FUNCTION_BLOCK BasicAdapter2 (* Basic FB with empty ECC *)
  (* Standard: 61499-2 *)
  (* Version 1.0, 2023-03-07, AK115394 *)
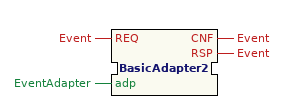
  EVENT_INPUT
    REQ;
  END_EVENT
  EVENT_OUTPUT
    CNF;
    RSP;
  END_EVENT
  SOCKETS
    adp : EventAdapter;
  END_SOCKETS
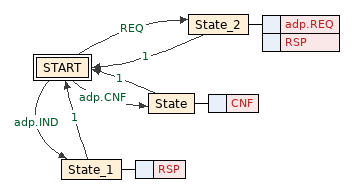
  EC_STATES
    START; (* Initial State *)
    State_2 : -> adp.REQ, -> RSP;
    State : -> CNF;
    State_1 : -> RSP;
  END_STATES
  EC_TRANSITIONS
    START TO State_2 := REQ;
    State_2 TO START := 1;
    START TO State := adp.CNF;
    START TO State_1 := adp.IND;
    State_1 TO START := 1;
    State TO START := 1;
  END_TRANSITIONS
END_FUNCTION_BLOCK
